(*
SPDX-FileCopyrightText: © 2026 Oleksandr Tiutyk <trofimich@gmail.com>
SPDX-License-Identifier: MIT
License: https://opensource.org/license/mit
*)

(*!
<summary>Selects the directions of hysteresis activation and reset.</summary>
<description>
Rising mode activates at or above the latch threshold and resets below the lower reset threshold. Falling mode
activates at or below the latch threshold and resets above the upper reset threshold.
</description>
*)
{attribute 'qualified_only'}
{attribute 'strict'}
{attribute 'to_string'}
TYPE HYSTERESIS_MODE :
(
    LATCH_ON_RISE_RESET_ON_FALL,
    LATCH_ON_FALL_RESET_ON_RISE
);
END_TYPE

(* stored: Version 1.1.0.1
   DUT HYSTERESIS_MODE: Id {003e51c0-c93b-4716-83a6-c87559b0eb6a} *)
